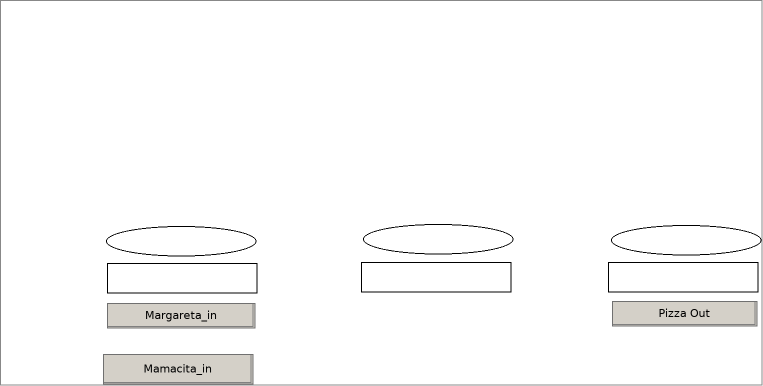
VISUALIZATION Visualization  // 763x386
    Rectangle (107,263 150x30)
    Rectangle (361,262 150x30)
    Rectangle (608,262 150x30)
    Button (107,303 148x25), "Margareta_in"
        tap MAIN.pizza_in
    Button (612,301 145x25), "Pizza Out"
        tap MAIN.pizza_out
    Ellipse (106,226 150x30), invisible if: NOT.MAIN.pizzaOven.PizzaOnDeck
    Ellipse (363,224 150x30), invisible if: NOT.MAIN.pizzaOven.PizzaInOven
    Ellipse (611,225 150x30), invisible if: NOT.MAIN.pizzaOven.PizzaDone
    Button (103,354 150x30), "Mamacita_in"
        tap MAIN.mamacita_in
END_VISUALIZATION

(* stored: Version 1.1.0.1, ProductVersion 3.1.4022.6
   Visu Visualization: Id {a2148bd0-893c-4d1a-bdec-3f3e76302e82} *)
